// TIA Portal V18 export
TYPE "PosList_IAI"
   STRUCT
      List : Array[0..39] of Struct
         Pos : Real;
         Vel : Int;
      END_STRUCT;
   END_STRUCT;
END_TYPE
